// TIA Portal V21 export
TYPE "OBJ_Analog_Type"
   STRUCT
      IO : Struct
         ix_Stop_Sim : Bool := true;
         iw_PEW : Int;
         if_PED : Real;
         ix_Reset : Bool;
         of_Value : Real;
         od_Value : DInt;
         oi_Value : Int;
         ox_Alarm : Bool;
      END_STRUCT;
      Data : Struct
         HMI : Struct
            x_Alarm : Bool;
            x_Simulation : Bool;
            x_Conf_Req : Bool;   // 1= Request Data Config From HMI
            d_Conf_Vis : DInt;   // Enable Visibility for Popup Config
            i_Nr_HMI_Vis : Int := 1;   // Univocal Number for HMI Visualization
            i_Req_Status : Int := 2;   // 0 = Forced Off 1 = Manual 2= Auto
            i_Real_Status : Int := 1;   // 1 = Off 2 = On 3 = Fault 4 = Forced On 5 = Forced Off
            f_Act_Value : Real;
            f_Man_Value : Real;
            f_Sim_Value : Real;
            "f_Compensation Value" : Real;   // Value for Offsetting the Block Exit Data
            f_Fault_Min_Val_In : Real;
            f_Fault_Max_Val_In : Real := 27648.0;
            f_Min_In : Real;
            f_Max_In : Real := 27648.0;
            f_Min_Out : Real;
            f_Max_Out : Real := 100.0;
            t_Time_Ton_Alm : Time := T#100MS;
         END_STRUCT;
         CFG : Struct
            i_Nr_HMI : Int := 1;   // Univocal Number for HMI Visualization
            i_Nr_Machine : Int := 0;
            "x_Use PED" : Bool := false;
            "x_Invert Measure" : Bool := false;   // Inversely Proportional Measure
            x_I_Or_O : Bool;   // 0= IN Value 1 = OUT Value
         END_STRUCT;
         SUP : Struct   // Logical Support
            x_AlwaysOff : Bool;
            x_Config_Edit : Bool;
            x_Aux_fp01 : Bool;
            x_Aux_fp02 : Bool;
            x_Aux_fp03 : Bool;
            x_Aux_fp04 : Bool;
            x_Aux_fp05 : Bool := false;
            x_Aux_fp06 : Bool := false;
            f_Value_In : Real;
            f_Max_Min_In : Real;
            f_Max_Min_Out : Real;
            f_Fact_K : Real;
            t_Ton_Alm : "OBJ_Timer_Type";
         END_STRUCT;
      END_STRUCT;
      ox_Status_Manual : Bool;   // ON if Valve in Manual
      ox_Status_Auto : Bool;   // ON if Valve in Automatic
   END_STRUCT;
END_TYPE
